(* CoDeSys 2.3.9.62 project: GUISmolPraktisk.pro *)
(* Libraries: SysLibTargetVisu.lib, Standard.lib, Iecsfc.lib 8.11.10 11:37:48, SYSLIBCALLBACK.LIB *)

(* PLC configuration (modules and I/O channels)
K-Bus [K_Bus] node 0, in %IB0 out %QB0
Internal Digital I/O [InternalDigIO] node 1, in %IB512 out %QB512
  Internal Digital Inputs [Internal_DIN] node 0, in %IB512 out %QB512
    DIN1 AT %IX2300.0 [BOOLOnX_I] Internal Digital Input Bit 1
    DIN2 AT %IX2300.1 [BOOLOnX_I] Internal Digital Input Bit 2
  Internal Digital Outputs [Internal_DOUT] node 1, in %IB513 out %QB512
    DOUT1 AT %QX2300.0 [BOOLOnX_Q] Internal Digital Output Bit 1
    DOUT2 AT %QX2300.1 [BOOLOnX_Q] Internal Digital Output Bit 2
Fieldbus variables [FB_VARS] node 3, in %IB0 out %QB0
Flag variables [FLAG_VARS] node 4, in %IB0 out %QB0
Modbus-Master [MB_MASTER] node 5, in %IB0 out %QB0
*)

(* Task configuration *)
TASK NewTask (PRIORITY := 15, INTERVAL := T#100ms);
	main();
END_TASK

(* Global variable list: Global_Variables *)
VAR_GLOBAL
	emergencyStopState : BOOL;

	tapPC : BOOL;
	pcTimer : INT;

	pedalsForward : BOOL;
	pedalsBack : BOOL;

	strenghtSlider : INT;

	innerOuterSlider : BOOL;
	innerOuterXOffset : INT;

	staticDynamicSlider : BOOL;
	staticDynamicXOffset : INT;
END_VAR

(* POU main, ST *)
PROGRAM main
VAR
	emergencyState : BOOL;
END_VAR
emergencyStopState := emergencyState;

innerOuterXOffset := 100 * BOOL_TO_INT(innerOuterSlider);
staticDynamicXOffset := 100 * BOOL_TO_INT(staticDynamicSlider);
END_PROGRAM

(* Visualisation GUISmol
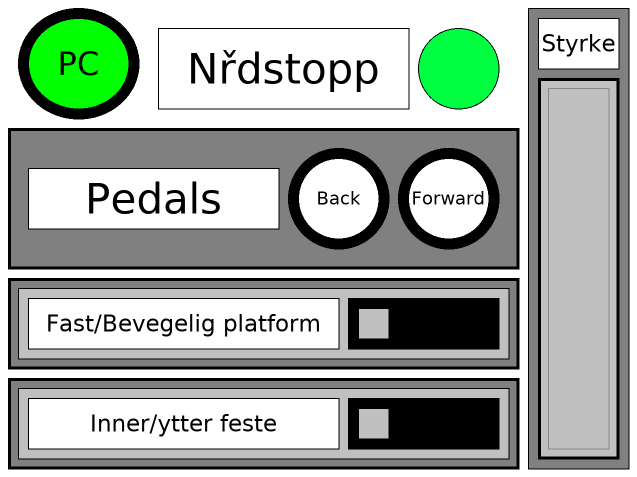
ellipse at (30,20)-(131,111): text "PC"; alarm colour if .tapPC; taps .tapPC
rounded rectangle at (30,170)-(281,231): text "Pedals"
ellipse at (300,160)-(381,241): text "Back"; alarm colour if .pedalsBack; taps .pedalsBack
ellipse at (410,160)-(491,241): text "Forward"; alarm colour if .pedalsForward; taps .pedalsForward
rounded rectangle at (540,20)-(621,71): text "Styrke"
rounded rectangle at (30,400)-(341,451): text "Inner/ytter feste"
rounded rectangle at (350,400)-(501,451): toggles .innerOuterSlider
rounded rectangle at (360,410)-(391,441): toggles .innerOuterSlider; x offset .innerOuterXOffset
rounded rectangle at (30,300)-(341,351): text "Fast/Bevegelig platform"
rounded rectangle at (350,300)-(501,351): toggles .staticDynamicSlider
rounded rectangle at (360,310)-(391,341): toggles .staticDynamicSlider; x offset .staticDynamicXOffset
rounded rectangle at (160,30)-(411,111): text "Nřdstopp"
ellipse at (420,30)-(501,111): alarm colour if .emergencyStopState
11 more shapes without text or variables
2 elements of other kinds (tables, trends, ...) not read
*)
